(* IEC 61131-3 sources: inproshop/Team-Test20_exported/OP70/1.Global, 7 files *)

(* ---- DB7000_Control.st ---- *)
VAR_GLOBAL
	Mode:Str_Mode;
	HMI:Str_HMI;
END_VAR
VAR_GLOBAL RETAIN PERSISTENT
	Machine AT %MB132516 : Str_Machine;
END_VAR

(* ---- DB7002_Recipe.st ---- *)
VAR_GLOBAL
END_VAR
VAR_GLOBAL RETAIN PERSISTENT

	RecipeChangePmt AT %MB133673 : BOOL;	//配方允许切换
	ParameterChangePmt AT %MB133674 : BOOL;	//参数允许更改
	RecipeNumTemp AT %MB133675 : INT;	//HMI选中还未保存到PLC的编号.
	RecipeNum AT %MB133677 : INT;	//配方元素编号.
	RecipeName AT %MB146778 : STRING(20);	//配方元素名称.
	RecipeNameTemp AT %MB179580 : STRING(20);	//HMI头部显示当前配方名称
	RecipeOk AT %MB133679 : BOOL;//配方可用
	DownLoad AT %MB133680 : BOOL;//配方下载
	TypeDataCur AT %MB327972 : Str_OP70_Recipe;//当前配方
	TypeData AT %MB490632 : ARRAY [0..10] OF Str_OP70_Recipe;//配方数据
END_VAR

(* ---- DB7003_Count.st ---- *)
VAR_GLOBAL RETAIN PERSISTENT
	Total AT %MB236200 : Str_Count;//总计数
	OK AT %MB236872 : Str_Count;//OK计数
	NG AT %MB237544 : Str_Count;//NG计数
END_VAR
VAR_GLOBAL
	Yield : REAL;//良品率
	Clear : BOOL;//清除计数
END_VAR

(* ---- DB7005_Communication.st ---- *)
VAR_GLOBAL
	TcpClient:ARRAY[0..9] OF Str_TcpClient;
	TcpSever:ARRAY[0..9] OF Str_TcpClient;
	From_OPXX AT %MW2000:Str_OP80_TO_OPXX;
	TO_OPXX AT %MW1000:Str_OPXX_TO_OP80;
	FromMaster AT %MW3000:Str_FromMaster;
END_VAR

(* ---- DB7050_DriveControl.st ---- *)
VAR_GLOBAL RETAIN PERSISTENT
	CylCtrl AT %MB436944 : ARRAY [0..63] OF Str_Cylinder;
	VacCtrl AT %MB445520 : ARRAY [0..63] OF Str_Cylinder;
	AxisCtrl AT %MB454096 : ARRAY [0..16] OF Str_Axis;
	Sensor AT %MB483336 : ARRAY [0..63] OF Str_Sensor;
	CamCtrl AT %MB337740 : ARRAY [0..1] OF Str_Cam;
	ESDCtrl AT %MB179360 : ARRAY [0..4] OF Str_ESD;
END_VAR

VAR_GLOBAL
	DoubleStart:ARRAY [1..3] OF Str_DoubleStart;
	Epson : ARRAY [1..10] OF Str_Epson;
	Kuka : ARRAY [1..10] OF Str_Kuka;
	Rotdisk:ARRAY [1..1] OF Str_Rotdisk;
	Stopper:ARRAY [1..20] OF Str_Stopper;
	Motor:ARRAY [1..10] OF Str_Motor;
	AI:ARRAY [1..200] OF Str_AI;
	GearCtrl:ARRAY [1..1] OF Str_Gear;
	AAS:ARRAY [1..1] OF Str_AAS;
	CodeCtrl:ARRAY [0..4] OF Str_Code;
	PrintCtrl:ARRAY [0..1] OF Str_Print;
	ScrewCtrl:ARRAY[0..4] OF Str_Screw;
END_VAR

(* ---- DB7070_Fault.st ---- *)
VAR_GLOBAL
	Estop:Str_OP70_FaultEstop;//紧急停止类报警
	Stop:Str_OP70_Faultstop;//暂停类报警
	Run:Str_OP70_FaultRun;//警告类报警
	EstopTotal:BOOL;//急停报警汇总
	StopTotal:BOOL;//暂停报警汇总
	RunTotal:BOOL;//警告汇总
END_VAR

(* ---- DB7090_Other.st ---- *)
VAR_GLOBAL RETAIN PERSISTENT
	{attribute 'ElemComment':='(),(人工上料位),(同步搬运1_1夹爪),(侧面1锁螺丝平台),(同步搬运1_2夹爪),(侧面2锁螺丝平台),(同步搬运2_1夹爪),(底面锁螺丝平台),(同步搬运2_2夹爪),(下料平台),()'}
	StationData AT %MB495384 : ARRAY [0..10] OF Str_OP70_StationData;

END_VAR
